// Mitsubishi GX Works2 project: plc_viet   PLC: Q00J

PROGRAM MAIN
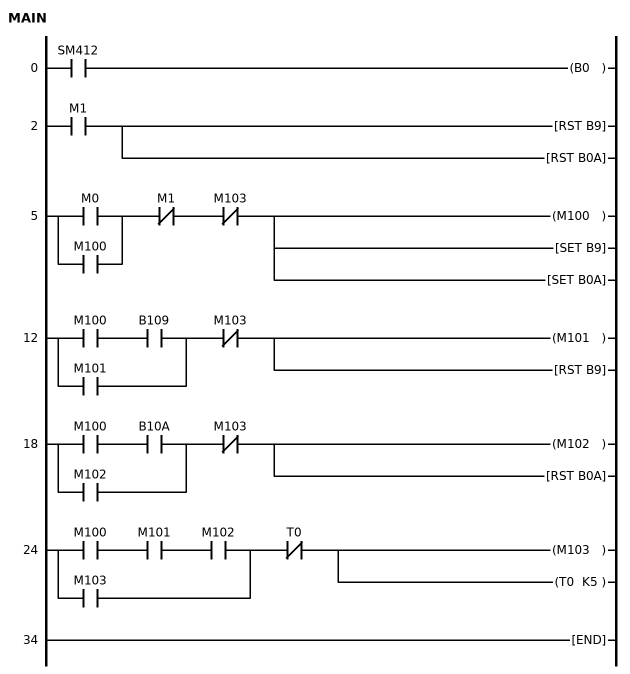
0     LD      SM412
      OUT     B0
2     LD      M1
      RST     B9
      RST     B0A
5     LD      M0
      OR      M100
      ANI     M1
      ANI     M103
      OUT     M100
      SET     B9
      SET     B0A
12    LD      M100
      AND     B109
      OR      M101
      ANI     M103
      OUT     M101
      RST     B9
18    LD      M100
      AND     B10A
      OR      M102
      ANI     M103
      OUT     M102
      RST     B0A
24    LD      M100
      AND     M101
      AND     M102
      OR      M103
      ANI     T0
      OUT     M103
      OUT     T0 K5
34    END
END_PROGRAM
